Fanuc KAREL source: GET_POS_TPE.kl

PROGRAM T
%NOLOCKGROUP
VAR
 v0 : INTEGER
 v1 : INTEGER
 v2 : INTEGER
 v3 : INTEGER
 res : XYZWPREXT
BEGIN
 res = GET_POS_TPE(v0, v1, v2, v3)
END T
